// TIA Portal V17 export
// export: Created 2024-08-09T12:53:21.3751551Z, ExportSetting WithDefaults, DisplayName Totally Integrated Automation Portal, DisplayVersion V17 Update 7, DisplayName TIA Portal Openness, DisplayVersion V17 Update 7, DisplayName TIA Portal Version Control Interface, DisplayVersion V17, DisplayName STEP 7 Professional, DisplayVersion V17 Update 7, DisplayName STEP 7 Safety, DisplayVersion V17 Update 6, DisplayName WinCC Professional, DisplayVersion V17 Update 7
TYPE "S_Info_Tour"
// stored: IsFailsafeCompliant false
   STRUCT
      _Camion { ExternalAccessible := 'False'; ExternalVisible := 'False'; ExternalWritable := 'False'} : String["T_CAMION"];   // code camion
      _ImmatCamion { ExternalAccessible := 'False'; ExternalVisible := 'False'; ExternalWritable := 'False'} : String["T_IMMAT"];   // Immatriculation camion
      _Chauffeur { ExternalAccessible := 'False'; ExternalVisible := 'False'; ExternalWritable := 'False'} : String["T_CHAUF"];   // code chauffeur
      _LbChauffeur { ExternalAccessible := 'False'; ExternalVisible := 'False'; ExternalWritable := 'False'} : String["T_CHAUF"];   // Libelle chauffeur
      _NoFeuilleRoute { ExternalAccessible := 'False'; ExternalVisible := 'False'; ExternalWritable := 'False'} : String["T_NO_TOUR"];   // no de feuille de route
      _NoTour { ExternalAccessible := 'False'; ExternalVisible := 'False'; ExternalWritable := 'False'} : String["T_NO_TOUR"];   // Numero de tour
      _Badge { ExternalAccessible := 'False'; ExternalVisible := 'False'; ExternalWritable := 'False'} : String["T_BADGE"];
      _NoLot { ExternalAccessible := 'False'; ExternalVisible := 'False'; ExternalWritable := 'False'} : String;
      _Tare { ExternalAccessible := 'False'; ExternalVisible := 'False'; ExternalWritable := 'False'} : Real;
      _PoidsMax { ExternalAccessible := 'False'; ExternalVisible := 'False'; ExternalWritable := 'False'} : Real;   // poids net maxi en charge du camion
      _PoidsVide { ExternalAccessible := 'False'; ExternalVisible := 'False'; ExternalWritable := 'False'} : Real;
      _IdTourn { ExternalAccessible := 'False'; ExternalVisible := 'False'; ExternalWritable := 'False'} : ULInt;
   END_STRUCT;
END_TYPE
